PROGRAM TEST_UNIT_VIRTUAL
VAR
	fbParent : RunUnitGeneric(ptBlock:= ADR(GVL.LOCAL_UNIT_CONTEXTS[1]));
	fbChild : RunUnitGeneric(ptBlock:= ADR(GVL.LOCAL_UNIT_CONTEXTS[2]));
	
	ptBlock : POINTER TO UnitBase := ADR(GVL.unitControls[2]);
	
	testCondition : bool ;
END_VAR

//the virtual station and coding example
fbParent(state=> );
fbChild(state=> );
//---------------------------

CASE fbChild.state OF
	0:
	// do next state
	ptBlock^.serialTransition := testCondition;
	1:
	//when transition condition meets , do next state
	IF ptBlock^.transitionByte = 16#3 THEN
		ptBlock^.serialTransition := TRUE;
	END_IF
	2..10:
		//try step mode
		ptBlock^.serialTransition :=TRUE;
	11:
	//direct set next state
	ptBlock^.nextState := 0;
	
	
END_CASE

END_PROGRAM

(* stored: Version 1.1.0.1, ProductVersion 3.1.4020.12
   POU TEST_UNIT_VIRTUAL: Id {def1cb56-2e92-494b-9c8e-90184f6eb8a7}, SpecialFunc None *)
